% RSLogix 500 project I2P JOB 09 - SOLUTION.RSS, saved by version 10.00.00.00 %
PROJECT "UNTITLED"    % processor: Bul.1763 MicroLogix 1100 Series B %

PROGRAM FILES
  LAD 2   4 rungs

DATA FILES
  O0 OUTPUT  4 elements
  I1 INPUT  6 elements
  S2 STATUS  66 elements
  B3 BINARY  1 elements
  T4 TIMER  1 elements
  C5 COUNTER  1 elements
  R6 CONTROL  1 elements
  N7 INTEGER  1 elements
  F8 FLOAT  1 elements

LADDER 2
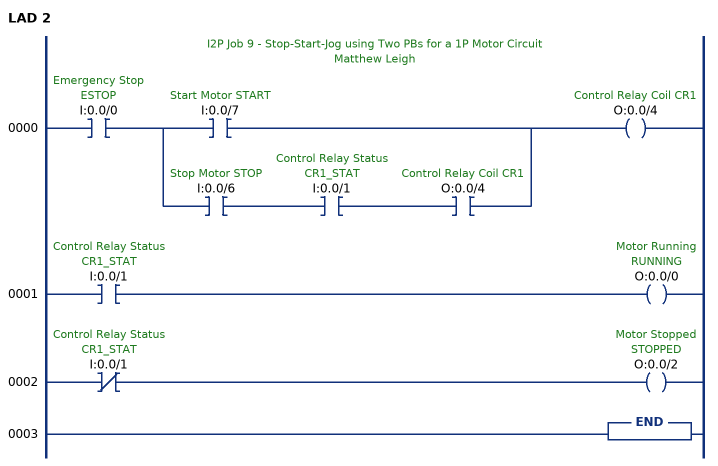
% Rung: 0 %
% I2P Job 9 - Stop-Start-Jog using Two PBs for a 1P Motor Circuit
% Matthew Leigh %
SOR XIC I:0.0/0 BST XIC I:0.0/7 NXB XIC I:0.0/6 XIC I:0.0/1 XIC O:0.0/4 BND OTE O:0.0/4 EOR
%   I:0.0/0  ESTOP  "Emergency Stop" %
%   I:0.0/7  START  "Start Motor" %
%   I:0.0/6  STOP  "Stop Motor" %
%   I:0.0/1  CR1_STAT  "Control Relay Status" %
%   O:0.0/4  CR1  "Control Relay Coil" %
% Rung: 1 %
SOR XIC I:0.0/1 OTE O:0.0/0 EOR
%   I:0.0/1  CR1_STAT  "Control Relay Status" %
%   O:0.0/0  RUNNING  "Motor Running" %
% Rung: 2 %
SOR XIO I:0.0/1 OTE O:0.0/2 EOR
%   I:0.0/1  CR1_STAT  "Control Relay Status" %
%   O:0.0/2  STOPPED  "Motor Stopped" %
% Rung: 3 %
SOR END EOR
